FUNCTION_BLOCK L1_Sensor

VAR_OUTPUT
	uiValue			: BOOL;					
END_VAR

VAR	
	hwValue AT %I*	: BOOL;					// Vinculación al hardware de la estación
	uiToolTip		: STRING;				// Tooltip en la visualización
END_VAR

METHOD ProcessCycle : BOOL
VAR_INPUT
	LocalHost	: BOOL;
END_VAR
VAR_OUTPUT
	sfcValue 	: BOOL;		// estado del sensor que se entregará al Grafcet
END_VAR
IF LocalHost THEN	
	hwValue := uiValue; 	// simulando la estación, el valor del sensor depende de la interfaz	
ELSE	
	uiValue := hwValue; 	// ejecutando en la estación, el valor de la visualización depende del hardware
END_IF
sfcValue := hwValue;		// estado del sensor que se entregará al Grafcet
END_METHOD

END_FUNCTION_BLOCK

(* stored: Version 1.1.0.1, ProductVersion 3.1.4024.11
   POU L1_Sensor: Id {c4029391-ebd0-4ae7-8ab5-3338cf1cc185}, SpecialFunc None
   Method ProcessCycle: Id {71ee41d9-0d14-4d00-a8c7-99dc223f0a9d} *)
